{attribute 'qualified_only'}
{attribute 'strict'}
TYPE E_MotorType :
(
	eLinear,
    eRotary,
    eStepper
);
END_TYPE

(* stored: Version 1.1.0.1, ProductVersion 3.1.4024.12
   DUT E_MotorType: Id {a227cca2-4e38-4aca-8f7b-ee72ec21358f} *)
